// SIMATIC S7-200 SMART project (STEP 7-Micro/WIN SMART), CPU SR20

SYMBOL_TABLE 表格 1
PH值              VD70
注肥桶号             VW10
注水桶号             VW12
循环桶号             VW14
灌溉标志             VW16
灌溉总水量            VD80
通道电磁阀1           VW20
通道电磁阀2           VW22
通道电磁阀3           VW24
通道电磁阀4           VW26
通道电磁阀5           VW28
母液目标流量1          VW30
母液目标流量2          VW32
母液目标流量3          VW34
母液目标流量4          VW36
母液目标流量5          VW38
母液注肥完成           VW40
液位高度1号桶          VW42
液位高度2号桶          VW44
液位高度3号桶          VW46
液位目标高度1          VW48
液位目标高度2          VW50
液位目标高度3          VW52
注清水完成            VW54
循环时长1号桶          VW56
循环时长2号桶          VW58
循环时长3号桶          VW60
排污标志             VW64
循环完成             VW62
EC值              VW68
END_SYMBOL_TABLE

SYMBOL_TABLE 系统符号
Always_On        SM0.0    // 始终接通
Clock_60s        SM0.4    // 针对 1 分钟的周期时间，时钟脉冲接通 30 s，断开 30 s.
Clock_1s         SM0.5    // 针对 1 s 的周期时间，时钟脉冲接通 0.5 s，断开 0.5 s.
END_SYMBOL_TABLE

ORGANIZATION_BLOCK MAIN:OB1
TITLE=程序注释
BEGIN
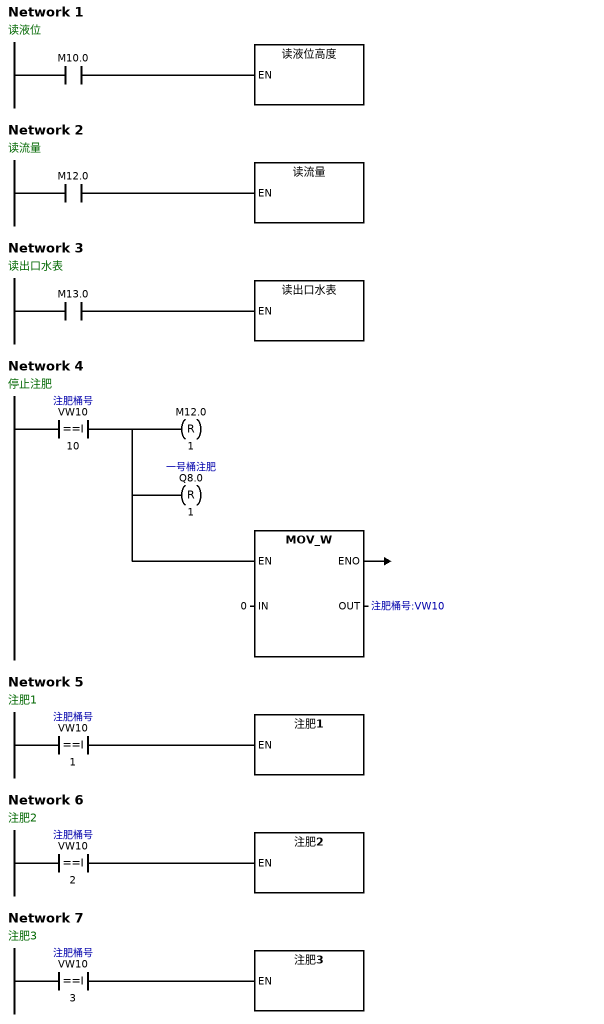
Network 1
// 读液位
LD     M10.0
CALL   读液位高度:SBR0
Network 2
// 读流量
LD     M12.0
CALL   读流量:SBR5
Network 3
// 读出口水表
LD     M13.0
CALL   读出口水表:SBR17
Network 4
// 停止注肥
LDW=   注肥桶号:VW10, 10
R      M12.0, 1
R      一号桶注肥:Q8.0, 1
MOVW   0, 注肥桶号:VW10
Network 5
// 注肥1
LDW=   注肥桶号:VW10, 1
CALL   注肥1:SBR6
Network 6
// 注肥2
LDW=   注肥桶号:VW10, 2
CALL   注肥2:SBR7
Network 7
// 注肥3
LDW=   注肥桶号:VW10, 3
CALL   注肥3:SBR8
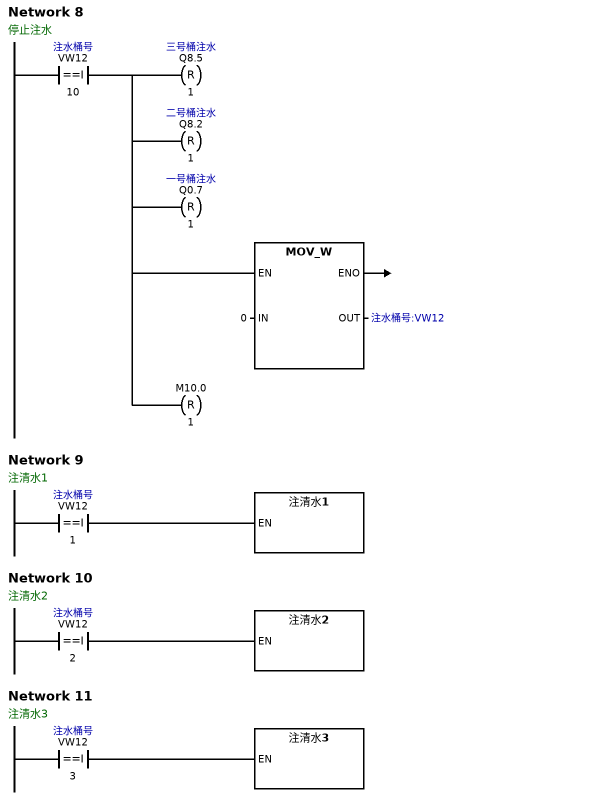
Network 8
// 停止注水
LDW=   注水桶号:VW12, 10
R      三号桶注水:Q8.5, 1
R      二号桶注水:Q8.2, 1
R      一号桶注水:Q0.7, 1
MOVW   0, 注水桶号:VW12
R      M10.0, 1
Network 9
// 注清水1
LDW=   注水桶号:VW12, 1
CALL   注清水1:SBR9
Network 10
// 注清水2
LDW=   注水桶号:VW12, 2
CALL   注清水2:SBR10
Network 11
// 注清水3
LDW=   注水桶号:VW12, 3
CALL   注清水3:SBR11
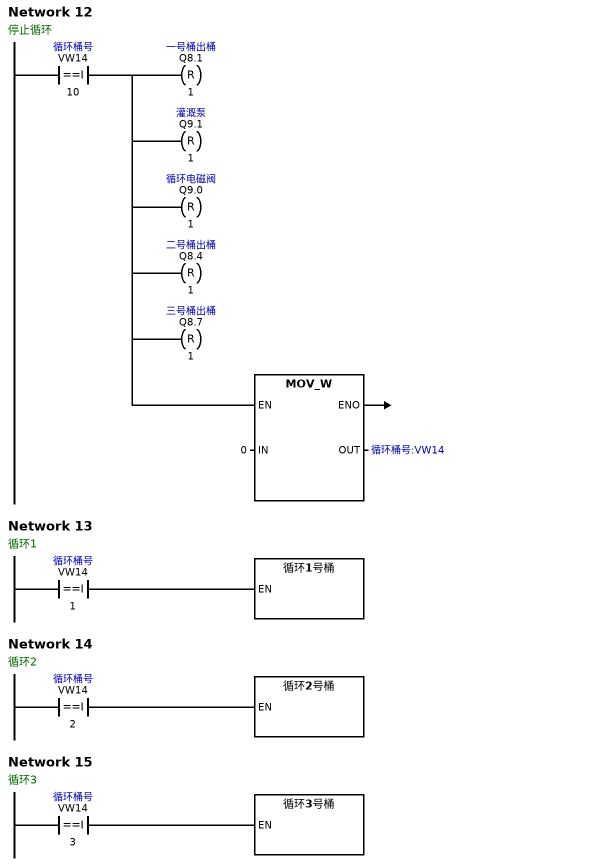
Network 12
// 停止循环
LDW=   循环桶号:VW14, 10
R      一号桶出桶:Q8.1, 1
R      灌溉泵:Q9.1, 1
R      循环电磁阀:Q9.0, 1
R      二号桶出桶:Q8.4, 1
R      三号桶出桶:Q8.7, 1
MOVW   0, 循环桶号:VW14
Network 13
// 循环1
LDW=   循环桶号:VW14, 1
CALL   循环1号桶:SBR12
Network 14
// 循环2
LDW=   循环桶号:VW14, 2
CALL   循环2号桶:SBR13
Network 15
// 循环3
LDW=   循环桶号:VW14, 3
CALL   循环3号桶:SBR14
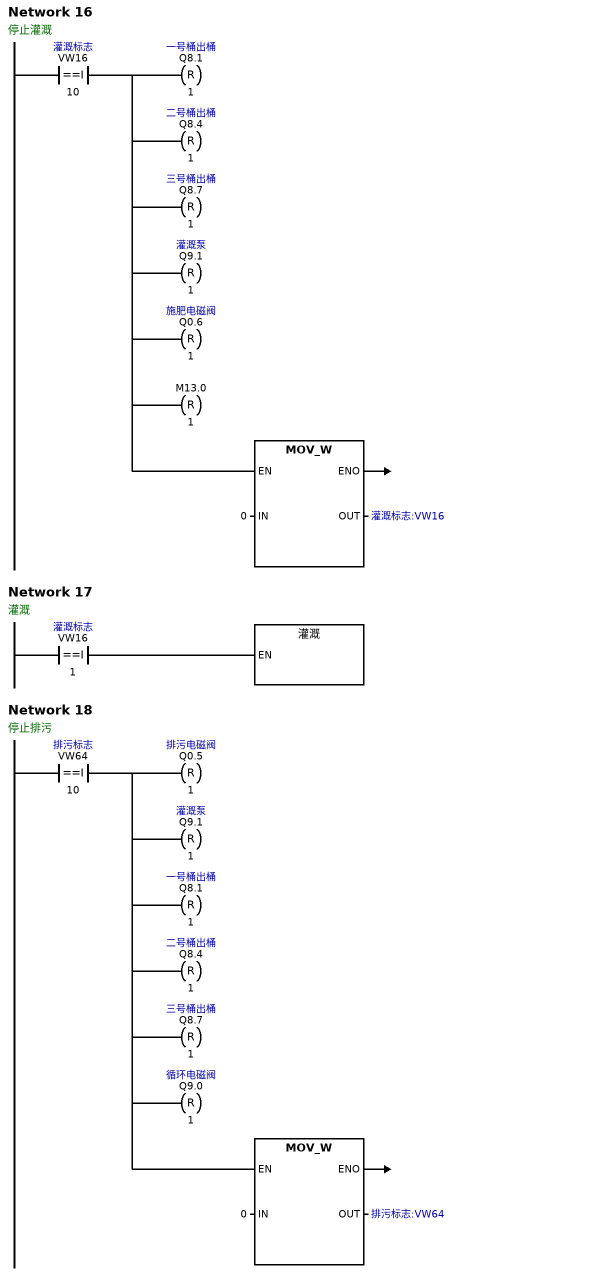
Network 16
// 停止灌溉
LDW=   灌溉标志:VW16, 10
R      一号桶出桶:Q8.1, 1
R      二号桶出桶:Q8.4, 1
R      三号桶出桶:Q8.7, 1
R      灌溉泵:Q9.1, 1
R      施肥电磁阀:Q0.6, 1
R      M13.0, 1
MOVW   0, 灌溉标志:VW16
Network 17
// 灌溉
LDW=   灌溉标志:VW16, 1
CALL   灌溉:SBR15
Network 18
// 停止排污
LDW=   排污标志:VW64, 10
R      排污电磁阀:Q0.5, 1
R      灌溉泵:Q9.1, 1
R      一号桶出桶:Q8.1, 1
R      二号桶出桶:Q8.4, 1
R      三号桶出桶:Q8.7, 1
R      循环电磁阀:Q9.0, 1
MOVW   0, 排污标志:VW64
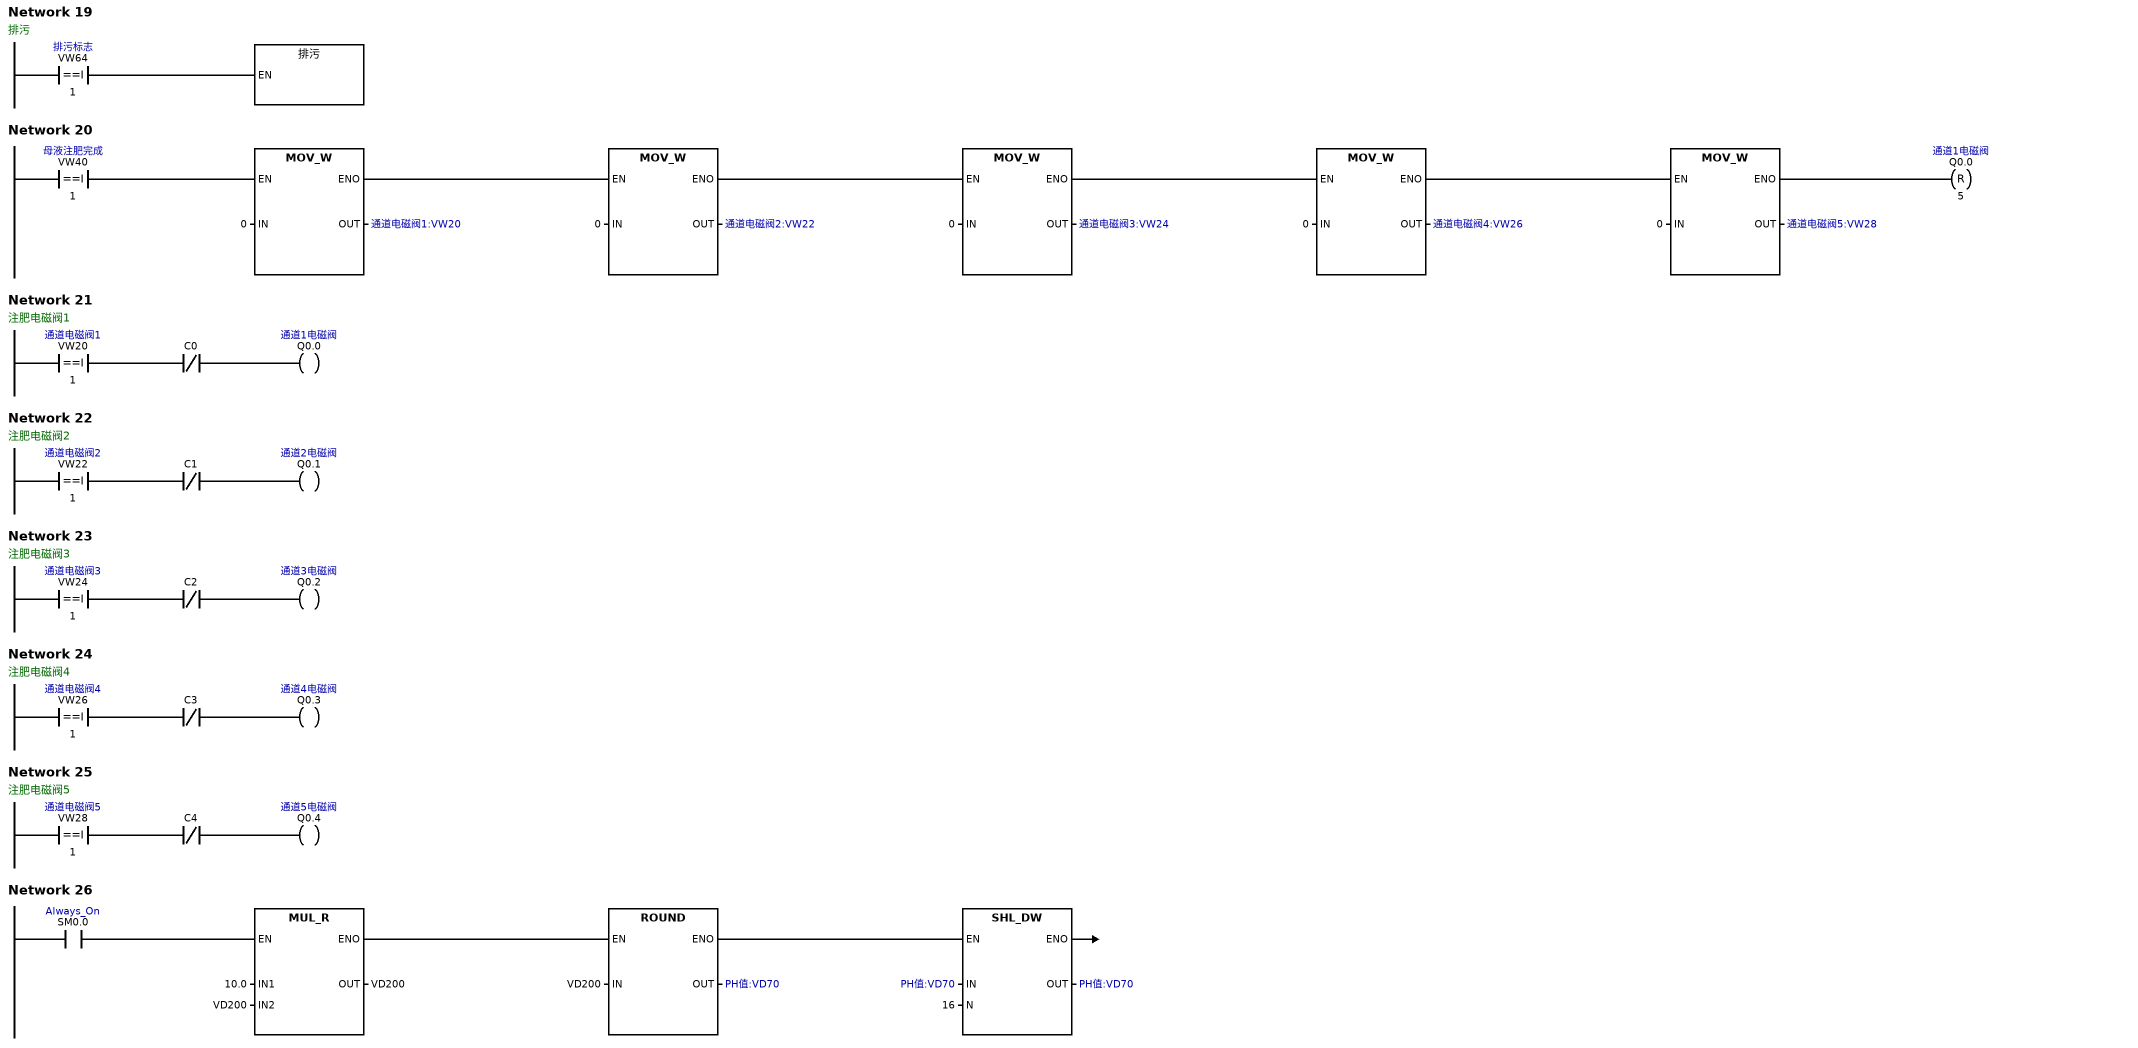
Network 19
// 排污
LDW=   排污标志:VW64, 1
CALL   排污:SBR16
Network 20
LDW=   母液注肥完成:VW40, 1
MOVW   0, 通道电磁阀1:VW20
AENO
MOVW   0, 通道电磁阀2:VW22
AENO
MOVW   0, 通道电磁阀3:VW24
AENO
MOVW   0, 通道电磁阀4:VW26
AENO
MOVW   0, 通道电磁阀5:VW28
AENO
R      通道1电磁阀:Q0.0, 5
Network 21
// 注肥电磁阀1
LDW=   通道电磁阀1:VW20, 1
AN     C0
=      通道1电磁阀:Q0.0
Network 22
// 注肥电磁阀2
LDW=   通道电磁阀2:VW22, 1
AN     C1
=      通道2电磁阀:Q0.1
Network 23
// 注肥电磁阀3
LDW=   通道电磁阀3:VW24, 1
AN     C2
=      通道3电磁阀:Q0.2
Network 24
// 注肥电磁阀4
LDW=   通道电磁阀4:VW26, 1
AN     C3
=      通道4电磁阀:Q0.3
Network 25
// 注肥电磁阀5
LDW=   通道电磁阀5:VW28, 1
AN     C4
=      通道5电磁阀:Q0.4
Network 26
LD     Always_On:SM0.0
*R     10.0, VD200
AENO
ROUND  VD200, PH值:VD70
AENO
SLD    PH值:VD70, 16
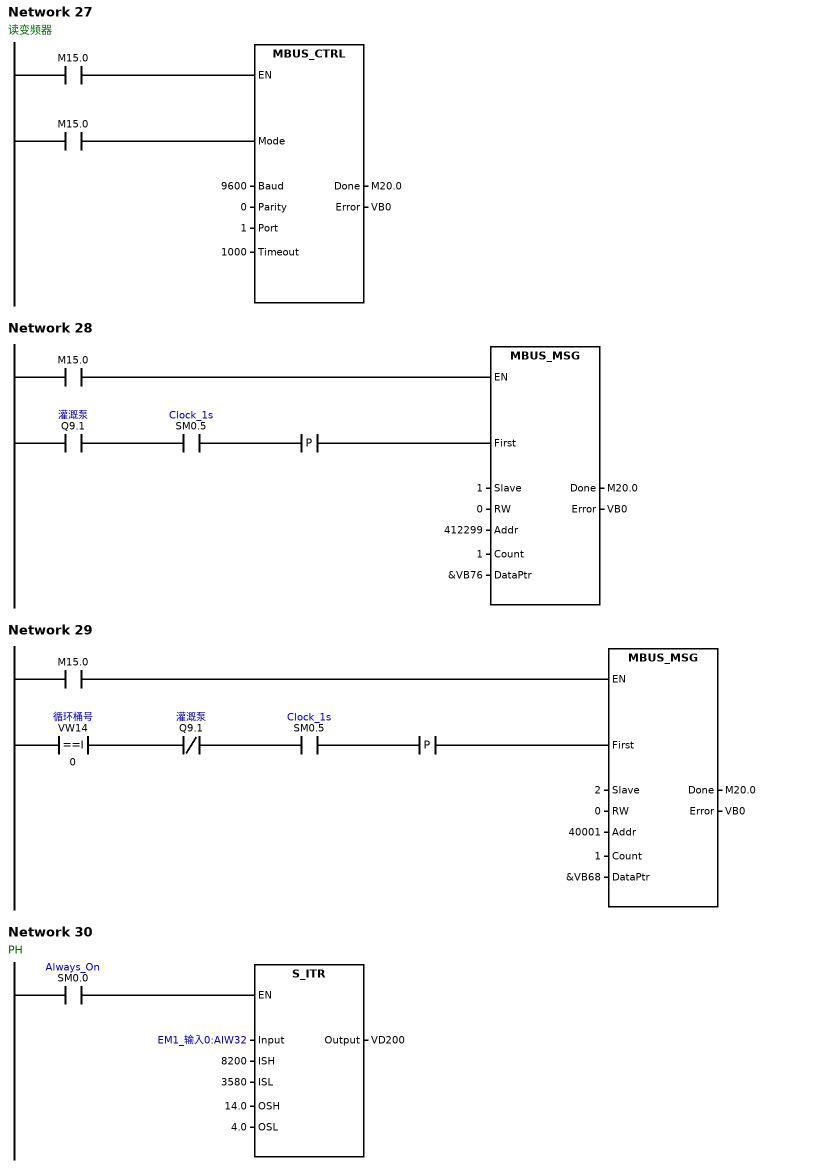
Network 27
// 读变频器
LD     M15.0
=      L60.0
LD     M15.0
=      L63.7
LD     L60.0
CALL   MBUS_CTRL:SBR1, L63.7, 9600, 0, 1, 1000, M20.0, VB0
Network 28
LD     M15.0
=      L60.0
LD     灌溉泵:Q9.1
A      Clock_1s:SM0.5
EU
=      L63.7
LD     L60.0
CALL   MBUS_MSG:SBR2, L63.7, 1, 0, 412299, 1, &VB76, M20.0, VB0
Network 29
LD     M15.0
=      L60.0
LDW=   循环桶号:VW14, 0
AN     灌溉泵:Q9.1
A      Clock_1s:SM0.5
EU
=      L63.7
LD     L60.0
CALL   MBUS_MSG:SBR2, L63.7, 2, 0, 40001, 1, &VB68, M20.0, VB0
Network 30
// PH
LD     Always_On:SM0.0
CALL   S_ITR:SBR18, EM1_输入0:AIW32, 8200, 3580, 14.0, 4.0, VD200
END_ORGANIZATION_BLOCK

SUBROUTINE_BLOCK 读液位高度:SBR0
TITLE=读液位高度
BEGIN
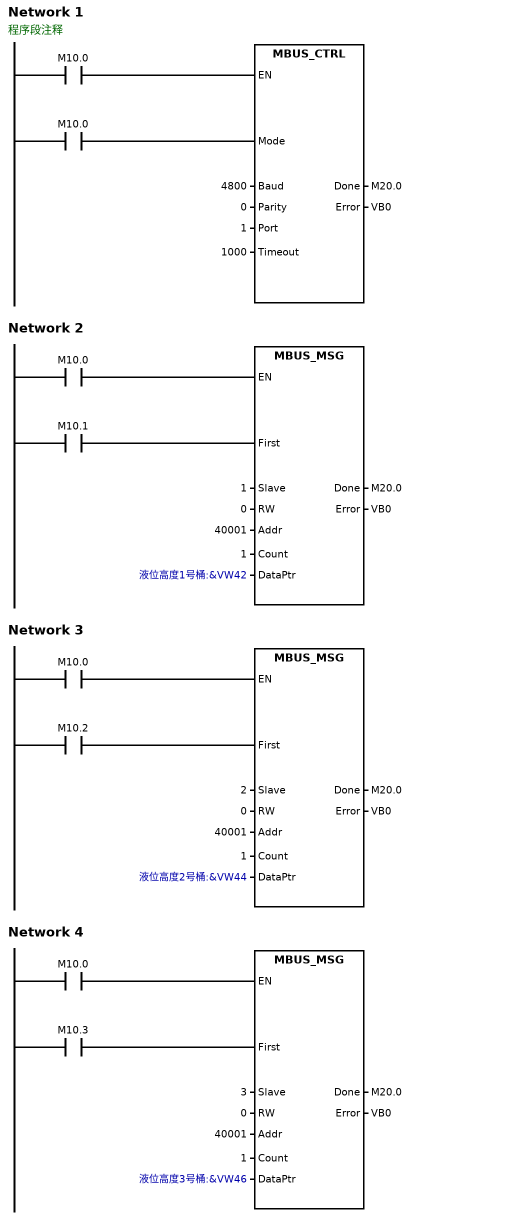
Network 1
// 程序段注释
LD     M10.0
=      L60.0
LD     M10.0
=      L63.7
LD     L60.0
CALL   MBUS_CTRL:SBR1, L63.7, 4800, 0, 1, 1000, M20.0, VB0
Network 2
LD     M10.0
=      L60.0
LD     M10.1
=      L63.7
LD     L60.0
CALL   MBUS_MSG:SBR2, L63.7, 1, 0, 40001, 1, &液位高度1号桶:VW42, M20.0, VB0
Network 3
LD     M10.0
=      L60.0
LD     M10.2
=      L63.7
LD     L60.0
CALL   MBUS_MSG:SBR2, L63.7, 2, 0, 40001, 1, &液位高度2号桶:VW44, M20.0, VB0
Network 4
LD     M10.0
=      L60.0
LD     M10.3
=      L63.7
LD     L60.0
CALL   MBUS_MSG:SBR2, L63.7, 3, 0, 40001, 1, &液位高度3号桶:VW46, M20.0, VB0
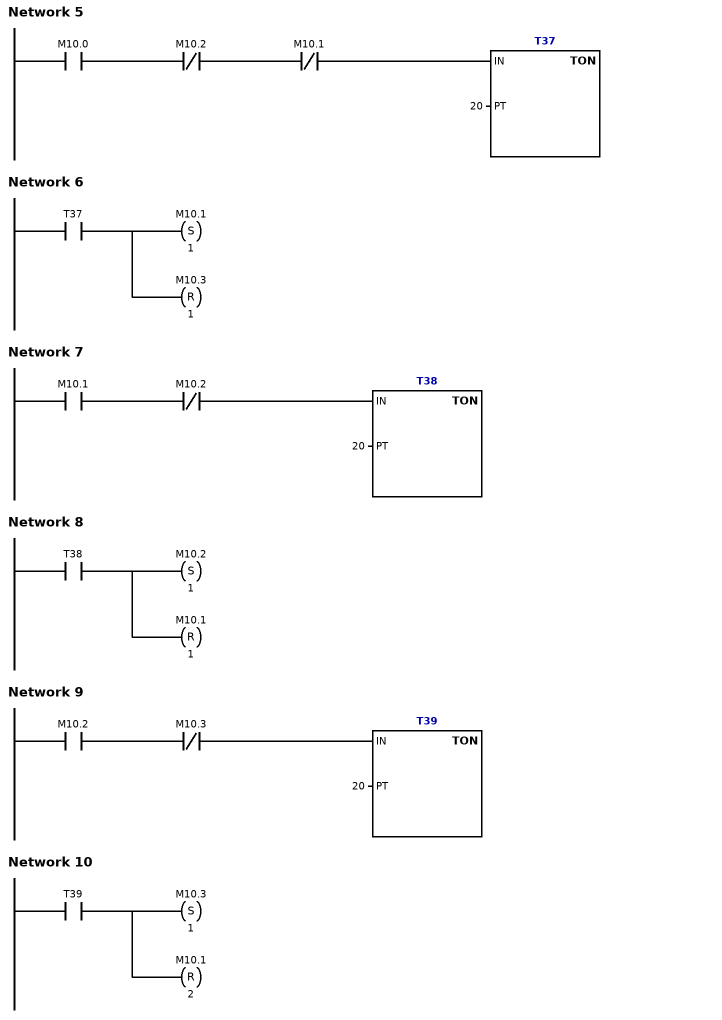
Network 5
LD     M10.0
AN     M10.2
AN     M10.1
TON    T37, 20
Network 6
LD     T37
S      M10.1, 1
R      M10.3, 1
Network 7
LD     M10.1
AN     M10.2
TON    T38, 20
Network 8
LD     T38
S      M10.2, 1
R      M10.1, 1
Network 9
LD     M10.2
AN     M10.3
TON    T39, 20
Network 10
LD     T39
S      M10.3, 1
R      M10.1, 2
Network 27
// 程序段注释
END_SUBROUTINE_BLOCK

// SBR1: protected block, not included

// SBR2: protected block, not included

// SBR3: protected block, not included

SUBROUTINE_BLOCK 读流量:SBR5
TITLE=子程序注释
BEGIN
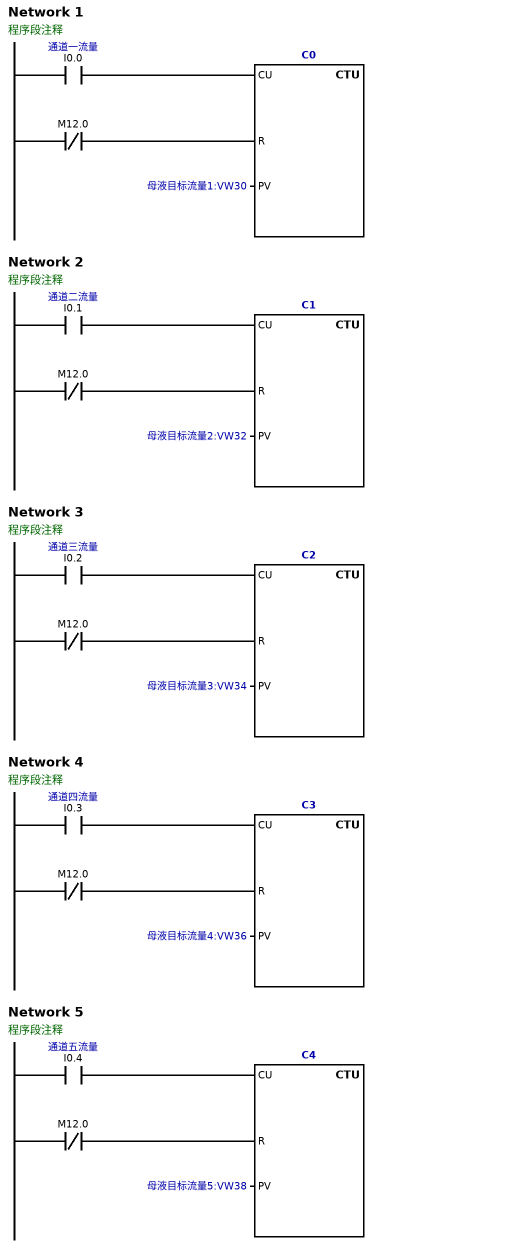
Network 1
// 程序段注释
LD     通道一流量:I0.0
LDN    M12.0
CTU    C0, 母液目标流量1:VW30
Network 2
// 程序段注释
LD     通道二流量:I0.1
LDN    M12.0
CTU    C1, 母液目标流量2:VW32
Network 3
// 程序段注释
LD     通道三流量:I0.2
LDN    M12.0
CTU    C2, 母液目标流量3:VW34
Network 4
// 程序段注释
LD     通道四流量:I0.3
LDN    M12.0
CTU    C3, 母液目标流量4:VW36
Network 5
// 程序段注释
LD     通道五流量:I0.4
LDN    M12.0
CTU    C4, 母液目标流量5:VW38
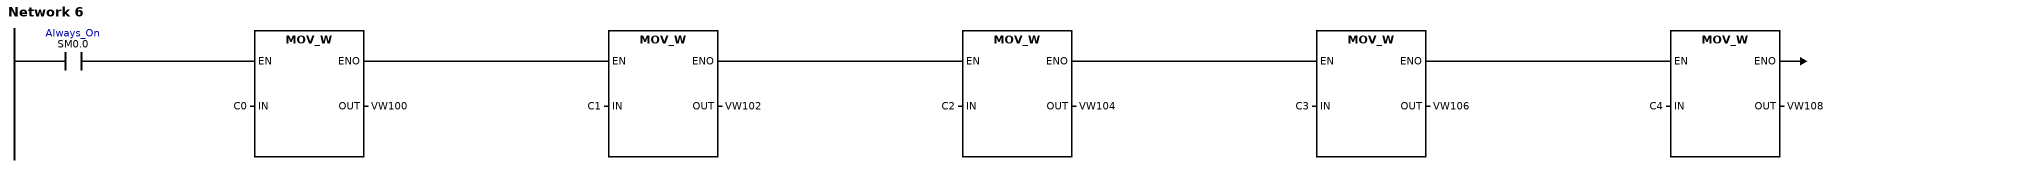
Network 6
LD     Always_On:SM0.0
MOVW   C0, VW100
AENO
MOVW   C1, VW102
AENO
MOVW   C2, VW104
AENO
MOVW   C3, VW106
AENO
MOVW   C4, VW108
END_SUBROUTINE_BLOCK

SUBROUTINE_BLOCK 注肥1:SBR6
TITLE=子程序注释
BEGIN
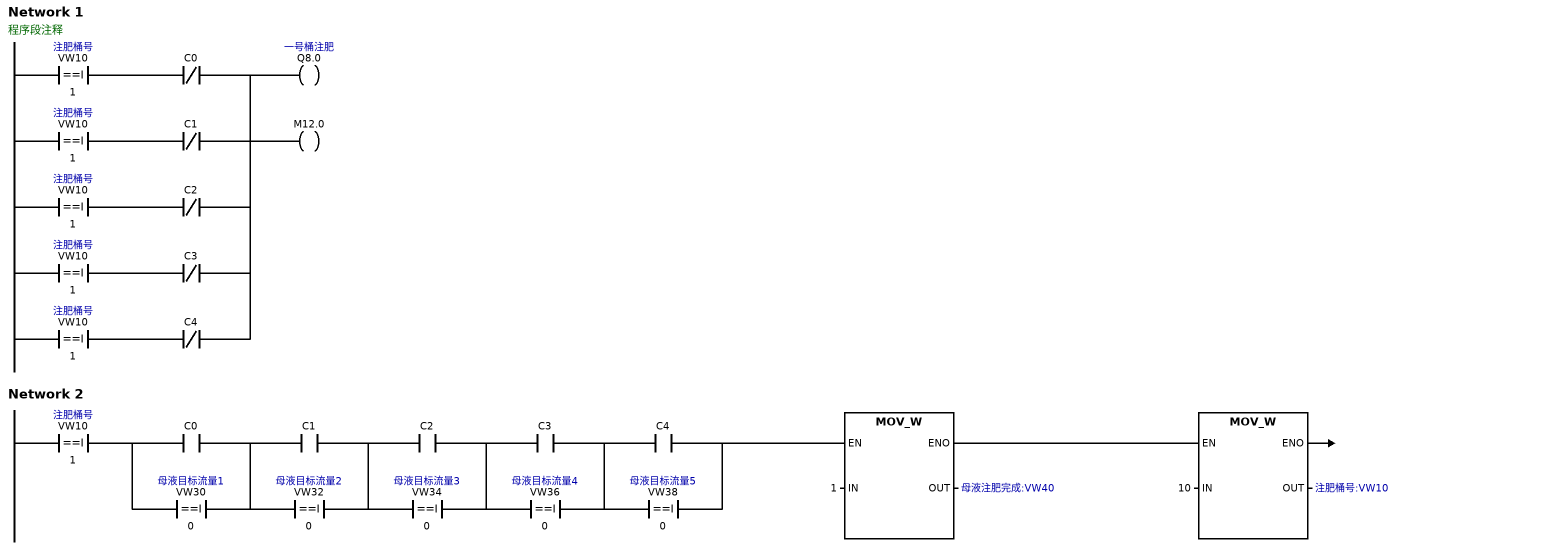
Network 1
// 程序段注释
LDW=   注肥桶号:VW10, 1
AN     C0
LDW=   注肥桶号:VW10, 1
AN     C1
OLD
LDW=   注肥桶号:VW10, 1
AN     C2
OLD
LDW=   注肥桶号:VW10, 1
AN     C3
OLD
LDW=   注肥桶号:VW10, 1
AN     C4
OLD
=      一号桶注肥:Q8.0
=      M12.0
Network 2
LDW=   注肥桶号:VW10, 1
LD     C0
OW=    母液目标流量1:VW30, 0
ALD
LD     C1
OW=    母液目标流量2:VW32, 0
ALD
LD     C2
OW=    母液目标流量3:VW34, 0
ALD
LD     C3
OW=    母液目标流量4:VW36, 0
ALD
LD     C4
OW=    母液目标流量5:VW38, 0
ALD
MOVW   1, 母液注肥完成:VW40
AENO
MOVW   10, 注肥桶号:VW10
END_SUBROUTINE_BLOCK

SUBROUTINE_BLOCK 注肥2:SBR7
TITLE=子程序注释
BEGIN
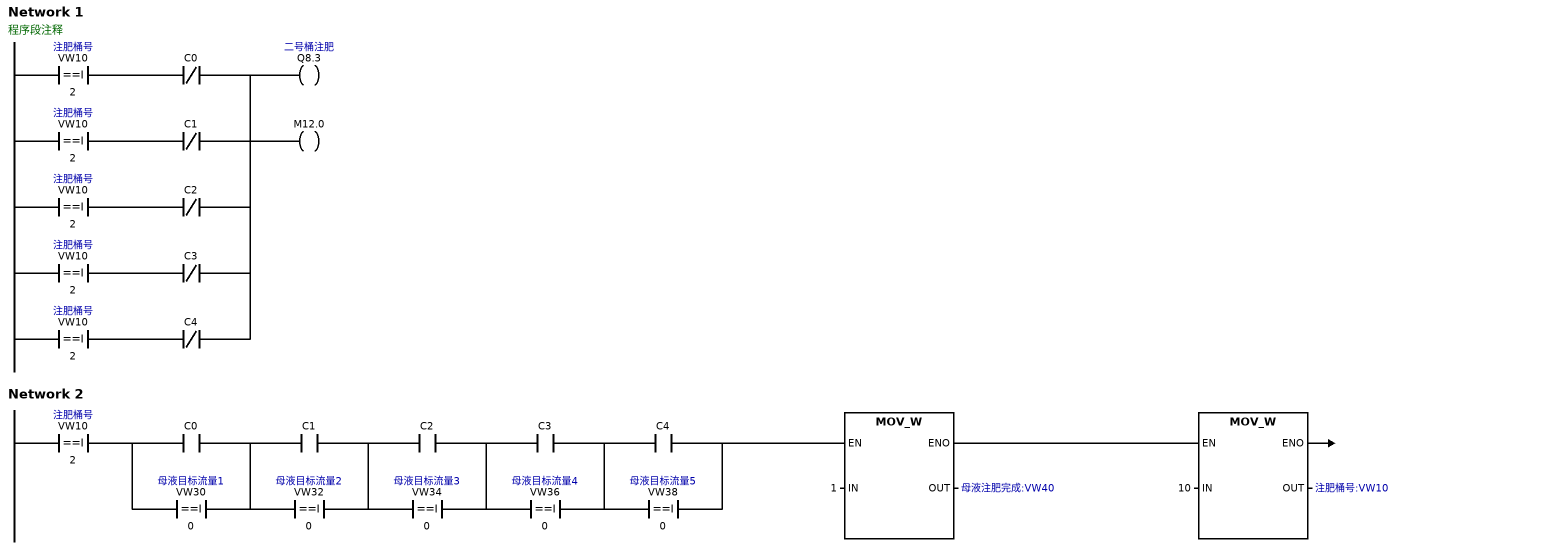
Network 1
// 程序段注释
LDW=   注肥桶号:VW10, 2
AN     C0
LDW=   注肥桶号:VW10, 2
AN     C1
OLD
LDW=   注肥桶号:VW10, 2
AN     C2
OLD
LDW=   注肥桶号:VW10, 2
AN     C3
OLD
LDW=   注肥桶号:VW10, 2
AN     C4
OLD
=      二号桶注肥:Q8.3
=      M12.0
Network 2
LDW=   注肥桶号:VW10, 2
LD     C0
OW=    母液目标流量1:VW30, 0
ALD
LD     C1
OW=    母液目标流量2:VW32, 0
ALD
LD     C2
OW=    母液目标流量3:VW34, 0
ALD
LD     C3
OW=    母液目标流量4:VW36, 0
ALD
LD     C4
OW=    母液目标流量5:VW38, 0
ALD
MOVW   1, 母液注肥完成:VW40
AENO
MOVW   10, 注肥桶号:VW10
END_SUBROUTINE_BLOCK

SUBROUTINE_BLOCK 注肥3:SBR8
TITLE=子程序注释
BEGIN
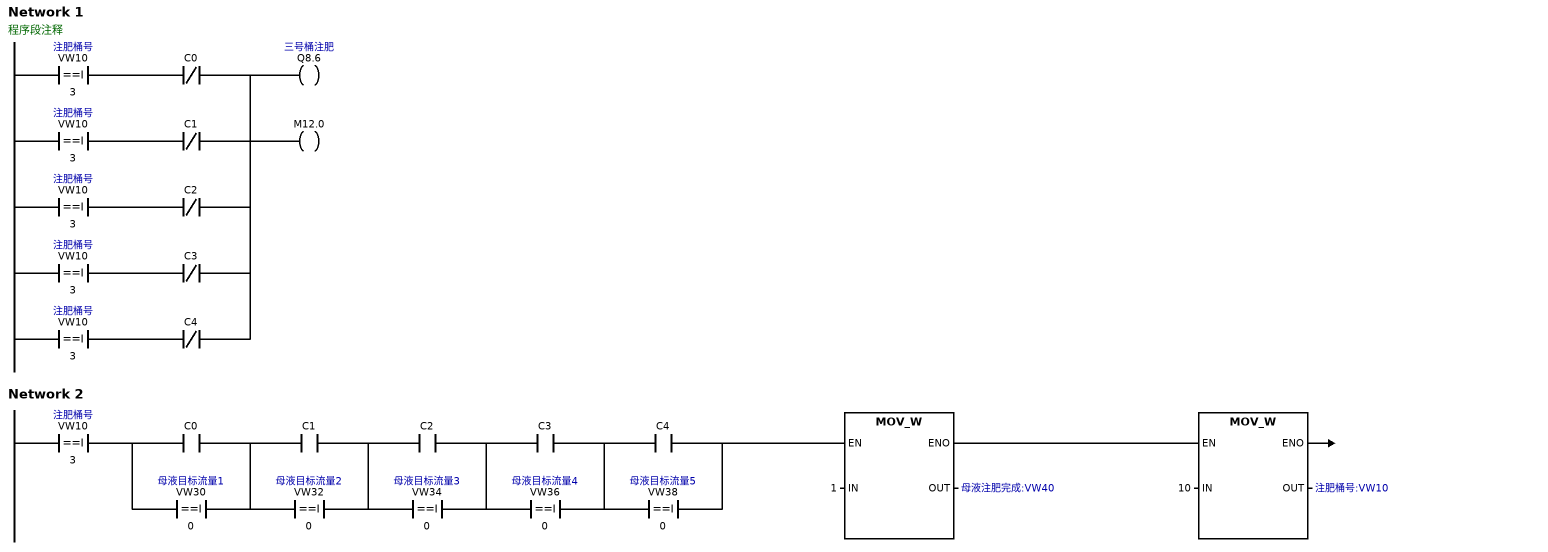
Network 1
// 程序段注释
LDW=   注肥桶号:VW10, 3
AN     C0
LDW=   注肥桶号:VW10, 3
AN     C1
OLD
LDW=   注肥桶号:VW10, 3
AN     C2
OLD
LDW=   注肥桶号:VW10, 3
AN     C3
OLD
LDW=   注肥桶号:VW10, 3
AN     C4
OLD
=      三号桶注肥:Q8.6
=      M12.0
Network 2
LDW=   注肥桶号:VW10, 3
LD     C0
OW=    母液目标流量1:VW30, 0
ALD
LD     C1
OW=    母液目标流量2:VW32, 0
ALD
LD     C2
OW=    母液目标流量3:VW34, 0
ALD
LD     C3
OW=    母液目标流量4:VW36, 0
ALD
LD     C4
OW=    母液目标流量5:VW38, 0
ALD
MOVW   1, 母液注肥完成:VW40
AENO
MOVW   10, 注肥桶号:VW10
END_SUBROUTINE_BLOCK

SUBROUTINE_BLOCK 注清水1:SBR9
TITLE=子程序注释
BEGIN
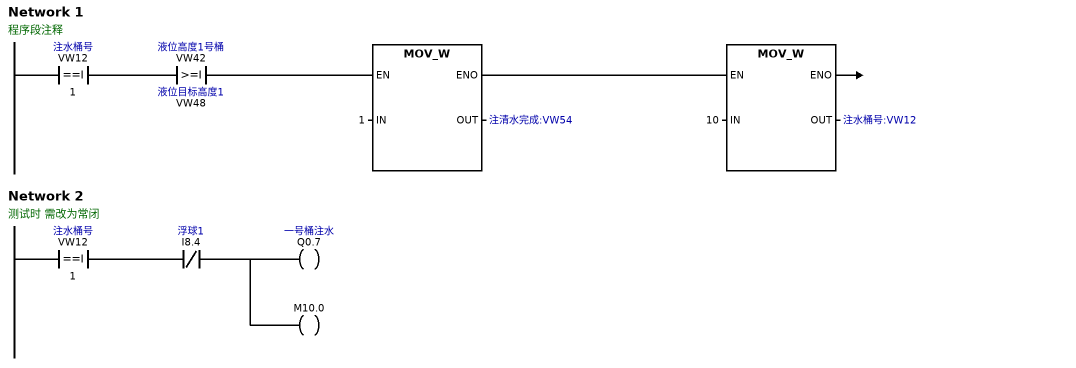
Network 1
// 程序段注释
LDW=   注水桶号:VW12, 1
AW>=   液位高度1号桶:VW42, 液位目标高度1:VW48
MOVW   1, 注清水完成:VW54
AENO
MOVW   10, 注水桶号:VW12
Network 2
// 测试时 需改为常闭
LDW=   注水桶号:VW12, 1
AN     浮球1:I8.4
=      一号桶注水:Q0.7
=      M10.0
END_SUBROUTINE_BLOCK

SUBROUTINE_BLOCK 注清水2:SBR10
TITLE=子程序注释
BEGIN
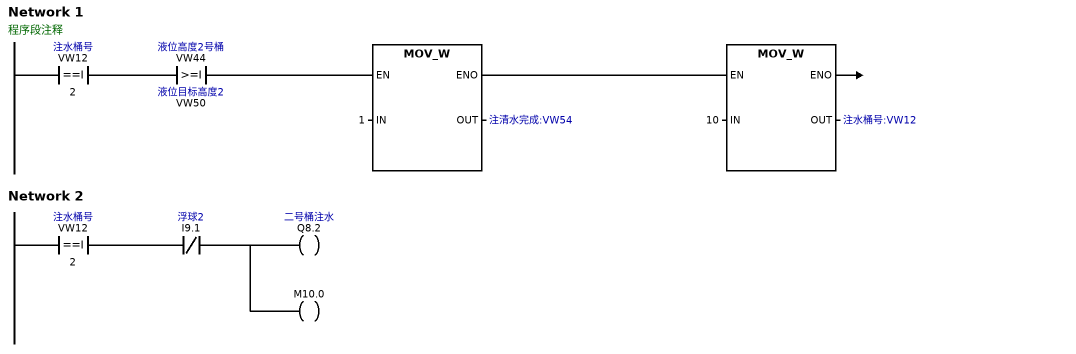
Network 1
// 程序段注释
LDW=   注水桶号:VW12, 2
AW>=   液位高度2号桶:VW44, 液位目标高度2:VW50
MOVW   1, 注清水完成:VW54
AENO
MOVW   10, 注水桶号:VW12
Network 2
LDW=   注水桶号:VW12, 2
AN     浮球2:I9.1
=      二号桶注水:Q8.2
=      M10.0
END_SUBROUTINE_BLOCK

SUBROUTINE_BLOCK 注清水3:SBR11
TITLE=子程序注释
BEGIN
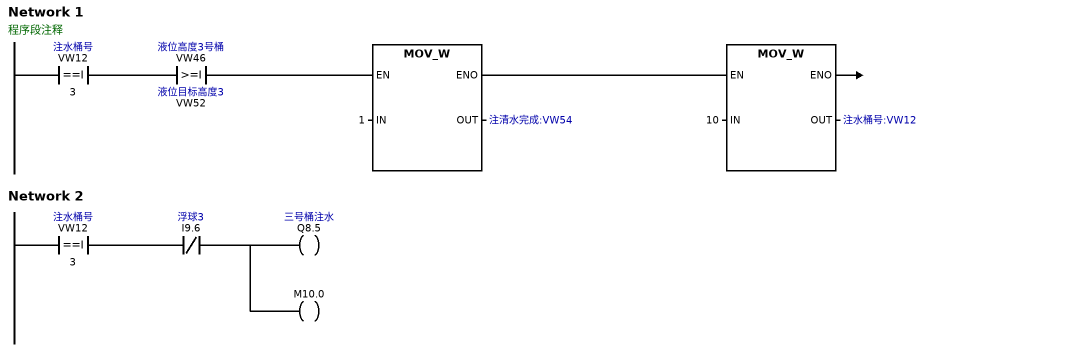
Network 1
// 程序段注释
LDW=   注水桶号:VW12, 3
AW>=   液位高度3号桶:VW46, 液位目标高度3:VW52
MOVW   1, 注清水完成:VW54
AENO
MOVW   10, 注水桶号:VW12
Network 2
LDW=   注水桶号:VW12, 3
AN     浮球3:I9.6
=      三号桶注水:Q8.5
=      M10.0
END_SUBROUTINE_BLOCK

SUBROUTINE_BLOCK 循环1号桶:SBR12
TITLE=子程序注释
BEGIN
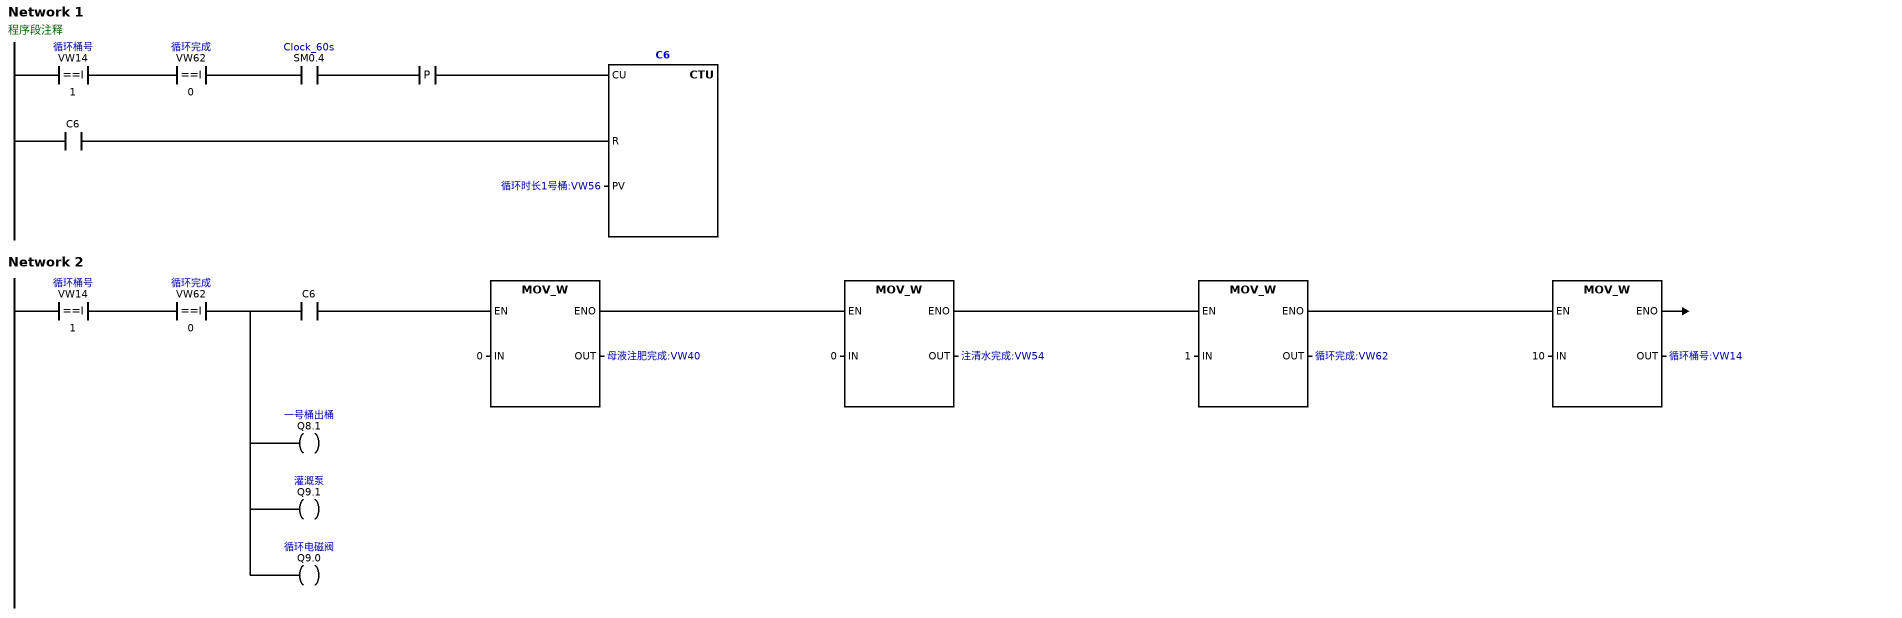
Network 1
// 程序段注释
LDW=   循环桶号:VW14, 1
AW=    循环完成:VW62, 0
A      Clock_60s:SM0.4
EU
LD     C6
CTU    C6, 循环时长1号桶:VW56
Network 2
LDW=   循环桶号:VW14, 1
AW=    循环完成:VW62, 0
LPS
A      C6
MOVW   0, 母液注肥完成:VW40
AENO
MOVW   0, 注清水完成:VW54
AENO
MOVW   1, 循环完成:VW62
AENO
MOVW   10, 循环桶号:VW14
LRD
=      一号桶出桶:Q8.1
LRD
=      灌溉泵:Q9.1
LPP
=      循环电磁阀:Q9.0
END_SUBROUTINE_BLOCK

SUBROUTINE_BLOCK 循环2号桶:SBR13
TITLE=子程序注释
BEGIN
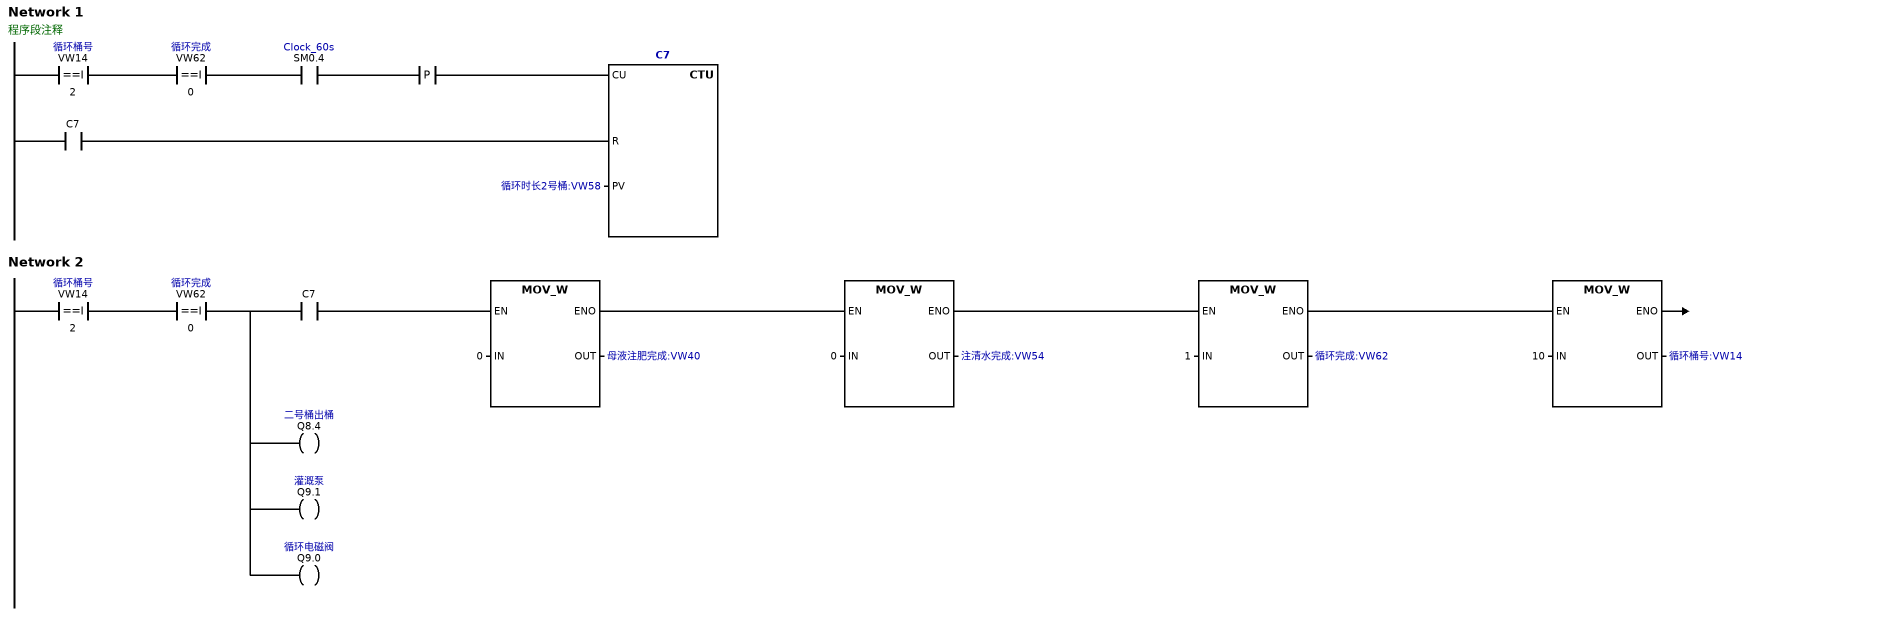
Network 1
// 程序段注释
LDW=   循环桶号:VW14, 2
AW=    循环完成:VW62, 0
A      Clock_60s:SM0.4
EU
LD     C7
CTU    C7, 循环时长2号桶:VW58
Network 2
LDW=   循环桶号:VW14, 2
AW=    循环完成:VW62, 0
LPS
A      C7
MOVW   0, 母液注肥完成:VW40
AENO
MOVW   0, 注清水完成:VW54
AENO
MOVW   1, 循环完成:VW62
AENO
MOVW   10, 循环桶号:VW14
LRD
=      二号桶出桶:Q8.4
LRD
=      灌溉泵:Q9.1
LPP
=      循环电磁阀:Q9.0
END_SUBROUTINE_BLOCK

SUBROUTINE_BLOCK 循环3号桶:SBR14
TITLE=子程序注释
BEGIN
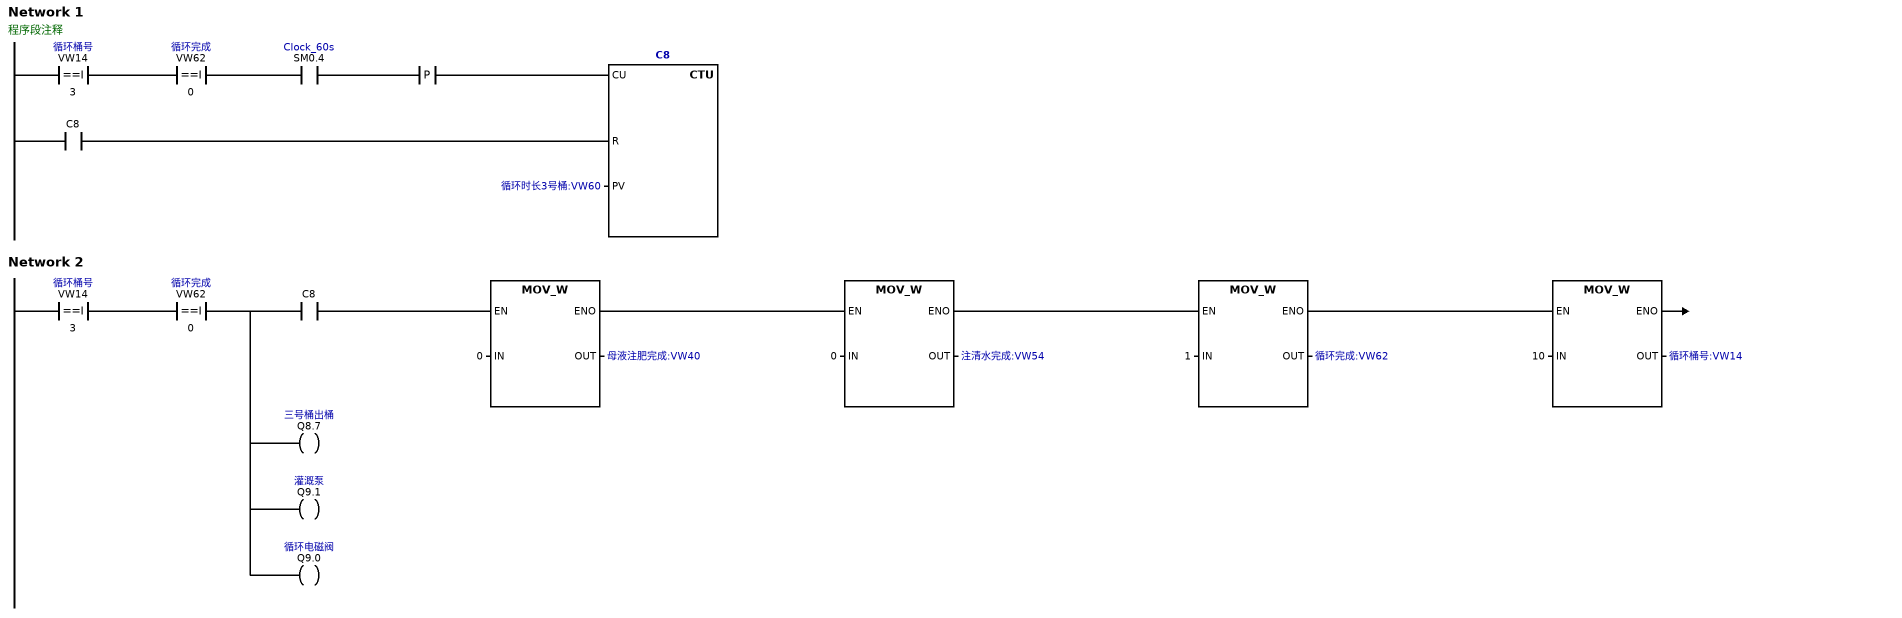
Network 1
// 程序段注释
LDW=   循环桶号:VW14, 3
AW=    循环完成:VW62, 0
A      Clock_60s:SM0.4
EU
LD     C8
CTU    C8, 循环时长3号桶:VW60
Network 2
LDW=   循环桶号:VW14, 3
AW=    循环完成:VW62, 0
LPS
A      C8
MOVW   0, 母液注肥完成:VW40
AENO
MOVW   0, 注清水完成:VW54
AENO
MOVW   1, 循环完成:VW62
AENO
MOVW   10, 循环桶号:VW14
LRD
=      三号桶出桶:Q8.7
LRD
=      灌溉泵:Q9.1
LPP
=      循环电磁阀:Q9.0
END_SUBROUTINE_BLOCK

SUBROUTINE_BLOCK 灌溉:SBR15
TITLE=子程序注释
BEGIN
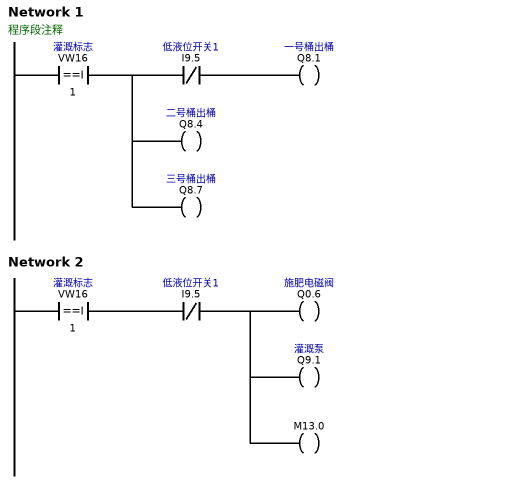
Network 1
// 程序段注释
LDW=   灌溉标志:VW16, 1
LPS
AN     低液位开关1:I9.5
=      一号桶出桶:Q8.1
LRD
=      二号桶出桶:Q8.4
LPP
=      三号桶出桶:Q8.7
Network 2
LDW=   灌溉标志:VW16, 1
AN     低液位开关1:I9.5
=      施肥电磁阀:Q0.6
=      灌溉泵:Q9.1
=      M13.0
END_SUBROUTINE_BLOCK

SUBROUTINE_BLOCK 排污:SBR16
TITLE=子程序注释
BEGIN
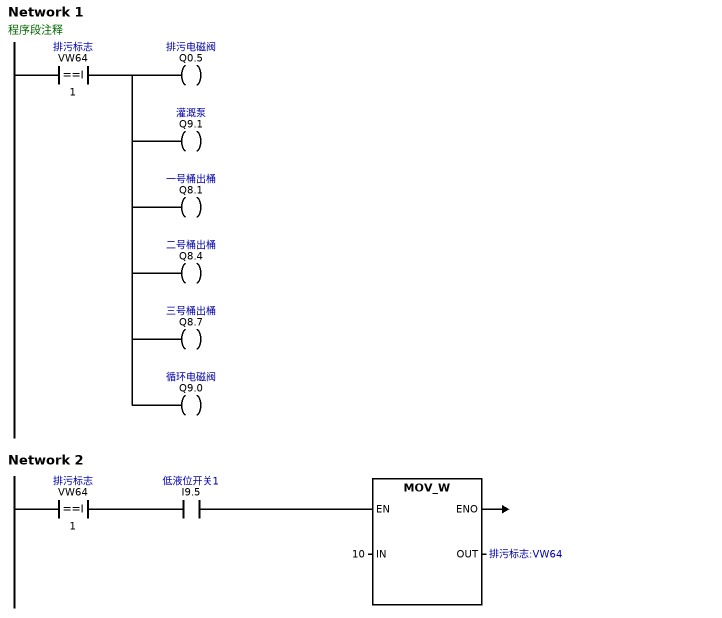
Network 1
// 程序段注释
LDW=   排污标志:VW64, 1
=      排污电磁阀:Q0.5
=      灌溉泵:Q9.1
=      一号桶出桶:Q8.1
=      二号桶出桶:Q8.4
=      三号桶出桶:Q8.7
=      循环电磁阀:Q9.0
Network 2
LDW=   排污标志:VW64, 1
A      低液位开关1:I9.5
MOVW   10, 排污标志:VW64
END_SUBROUTINE_BLOCK

SUBROUTINE_BLOCK 读出口水表:SBR17
TITLE=子程序注释
BEGIN
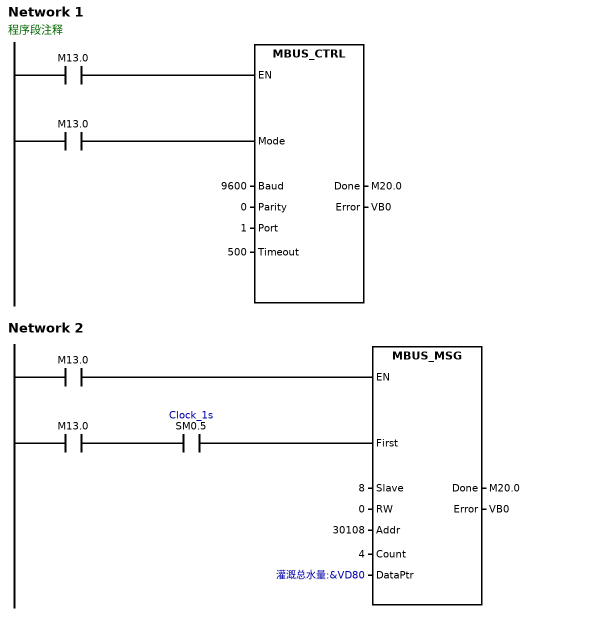
Network 1
// 程序段注释
LD     M13.0
=      L60.0
LD     M13.0
=      L63.7
LD     L60.0
CALL   MBUS_CTRL:SBR1, L63.7, 9600, 0, 1, 500, M20.0, VB0
Network 2
LD     M13.0
=      L60.0
LD     M13.0
A      Clock_1s:SM0.5
=      L63.7
LD     L60.0
CALL   MBUS_MSG:SBR2, L63.7, 8, 0, 30108, 4, &灌溉总水量:VD80, M20.0, VB0
END_SUBROUTINE_BLOCK

// SBR18: protected block, not included
